// TIA Portal V19 export
TYPE "CTRL_ADIN"
   STRUCT
      status : Bool := false;
      sim : "UDT_SIM_BOOL";
   END_STRUCT;
END_TYPE
